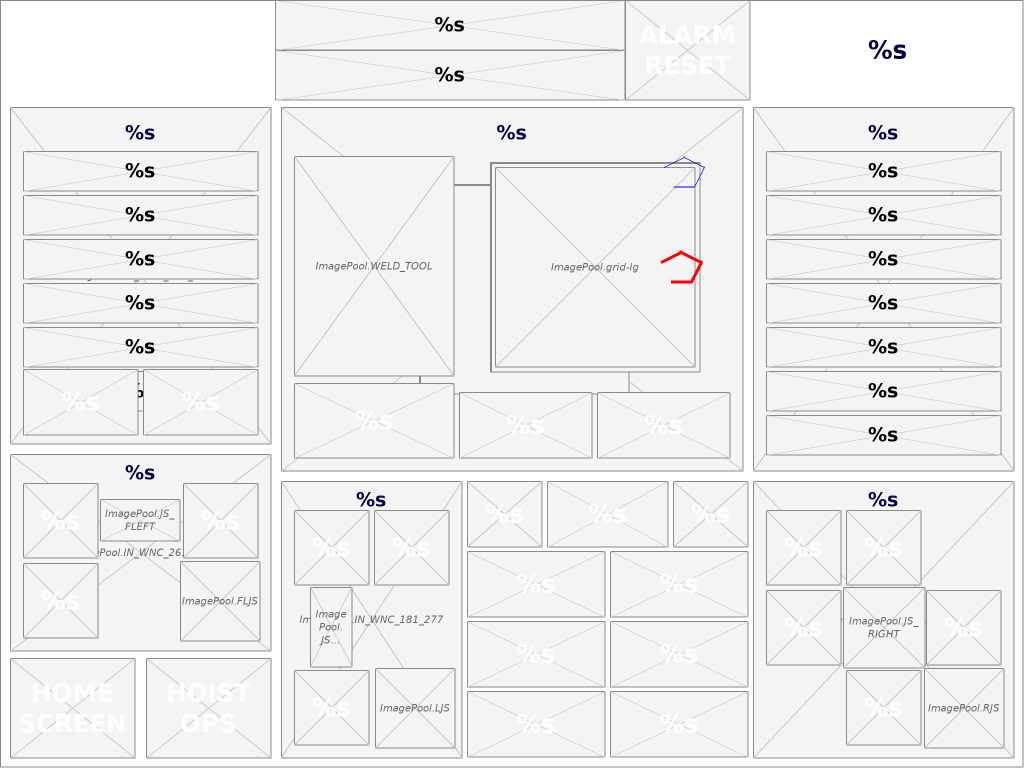
VISUALIZATION TOOL_OPS_SCREEN  // 1024x768, background image ImagePool.background1
    Image (281,107 462x364), image: ImagePool.IN_WNC_462_364
    Group (419,184 70x70), invisible if: MAIN.Visualization.P14_SMALL_PIE_DISPLAY_INVISIBLE
        Pie (1,1 209x209), invisible if: MAIN.RGP.PROG.P14_PIE_INVISIBLE[0]
        Pie (1,1 209x209), invisible if: MAIN.RGP.PROG.P14_PIE_INVISIBLE[1]
            p426801730: MAIN.RGP.PROG.P14_PIE_BEGIN[1]
            p2124672552: MAIN.RGP.PROG.P14_PIE_END[1]
        Pie (1,1 209x209), invisible if: MAIN.RGP.PROG.P14_PIE_INVISIBLE[2]
            p426801730: MAIN.RGP.PROG.P14_PIE_BEGIN[2]
            p2124672552: MAIN.RGP.PROG.P14_PIE_END[2]
        Pie (1,1 209x209), invisible if: MAIN.RGP.PROG.P14_PIE_INVISIBLE[3]
            p426801730: MAIN.RGP.PROG.P14_PIE_BEGIN[3]
            p2124672552: MAIN.RGP.PROG.P14_PIE_END[3]
        Pie (1,1 209x209), invisible if: MAIN.RGP.PROG.P14_PIE_INVISIBLE[4]
            p426801730: MAIN.RGP.PROG.P14_PIE_BEGIN[4]
            p2124672552: MAIN.RGP.PROG.P14_PIE_END[4]
        Pie (1,1 209x209), invisible if: MAIN.RGP.PROG.P14_PIE_INVISIBLE[5]
            p426801730: MAIN.RGP.PROG.P14_PIE_BEGIN[5]
            p2124672552: MAIN.RGP.PROG.P14_PIE_END[5]
        Pie (1,1 209x209), invisible if: MAIN.RGP.PROG.P14_PIE_INVISIBLE[6]
            p426801730: MAIN.RGP.PROG.P14_PIE_BEGIN[6]
            p2124672552: MAIN.RGP.PROG.P14_PIE_END[6]
        Pie (1,1 209x209), invisible if: MAIN.RGP.PROG.P14_PIE_INVISIBLE[7]
            p426801730: MAIN.RGP.PROG.P14_PIE_BEGIN[7]
            p2124672552: MAIN.RGP.PROG.P14_PIE_END[7]
        Pie (1,1 209x209), invisible if: MAIN.RGP.PROG.P14_PIE_INVISIBLE[8]
            p426801730: MAIN.RGP.PROG.P14_PIE_BEGIN[8]
            p2124672552: MAIN.RGP.PROG.P14_PIE_END[8]
        Pie (1,1 209x209), invisible if: MAIN.RGP.PROG.P14_PIE_INVISIBLE[9]
            p426801730: MAIN.RGP.PROG.P14_PIE_BEGIN[9]
            p2124672552: MAIN.RGP.PROG.P14_PIE_END[9]
        Pie (1,1 209x209), invisible if: MAIN.RGP.PROG.P14_PIE_INVISIBLE[10]
            p426801730: MAIN.RGP.PROG.P14_PIE_BEGIN[10]
            p2124672552: MAIN.RGP.PROG.P14_PIE_END[10]
        Pie (1,1 209x209), invisible if: MAIN.RGP.PROG.P14_PIE_INVISIBLE[11]
            p426801730: MAIN.RGP.PROG.P14_PIE_BEGIN[11]
            p2124672552: MAIN.RGP.PROG.P14_PIE_END[11]
        Pie (1,1 209x209), invisible if: MAIN.RGP.PROG.P14_PIE_INVISIBLE[12]
            p426801730: MAIN.RGP.PROG.P14_PIE_BEGIN[12]
            p2124672552: MAIN.RGP.PROG.P14_PIE_END[12]
        Pie (1,1 209x209), invisible if: MAIN.RGP.PROG.P14_PIE_INVISIBLE[13]
            p426801730: MAIN.RGP.PROG.P14_PIE_BEGIN[13]
            p2124672552: MAIN.RGP.PROG.P14_PIE_END[13]
        Pie (1,1 209x209), invisible if: MAIN.RGP.PROG.P14_PIE_INVISIBLE[14]
            p426801730: MAIN.RGP.PROG.P14_PIE_BEGIN[14]
            p2124672552: MAIN.RGP.PROG.P14_PIE_END[14]
        Pie (1,1 209x209), invisible if: MAIN.RGP.PROG.P14_PIE_INVISIBLE[15]
            p426801730: MAIN.RGP.PROG.P14_PIE_BEGIN[15]
            p2124672552: MAIN.RGP.PROG.P14_PIE_END[15]
        Pie (0,0 210x210), invisible if: MAIN.RGP.PROG.P14_PIE_INVISIBLE[16]
            p426801730: MAIN.RGP.PROG.P14_PIE_BEGIN[16]
            p2124672552: MAIN.RGP.PROG.P14_PIE_END[16]
        Pie (1,1 209x209), invisible if: MAIN.RGP.PROG.P14_PIE_INVISIBLE[17]
            p426801730: MAIN.RGP.PROG.P14_PIE_BEGIN[17]
            p2124672552: MAIN.RGP.PROG.P14_PIE_END[17]
        Pie (1,1 209x209), invisible if: MAIN.RGP.PROG.P14_PIE_INVISIBLE[18]
            p426801730: MAIN.RGP.PROG.P14_PIE_BEGIN[18]
            p2124672552: MAIN.RGP.PROG.P14_PIE_END[18]
        Pie (1,1 209x209), invisible if: MAIN.RGP.PROG.P14_PIE_INVISIBLE[19]
            p426801730: MAIN.RGP.PROG.P14_PIE_BEGIN[19]
            p2124672552: MAIN.RGP.PROG.P14_PIE_END[19]
        Pie (1,1 209x209), invisible if: MAIN.RGP.PROG.P14_PIE_INVISIBLE[20]
            p426801730: MAIN.RGP.PROG.P14_PIE_BEGIN[20]
            p2124672552: MAIN.RGP.PROG.P14_PIE_END[20]
        Pie (1,1 209x209), invisible if: MAIN.RGP.PROG.P14_PIE_INVISIBLE[21]
            p426801730: MAIN.RGP.PROG.P14_PIE_BEGIN[21]
            p2124672552: MAIN.RGP.PROG.P14_PIE_END[21]
        Pie (1,1 209x209), invisible if: MAIN.RGP.PROG.P14_PIE_INVISIBLE[22]
            p426801730: MAIN.RGP.PROG.P14_PIE_BEGIN[22]
            p2124672552: MAIN.RGP.PROG.P14_PIE_END[22]
        Pie (1,1 209x209), invisible if: MAIN.RGP.PROG.P14_PIE_INVISIBLE[23]
            p426801730: MAIN.RGP.PROG.P14_PIE_BEGIN[23]
            p2124672552: MAIN.RGP.PROG.P14_PIE_END[23]
        Pie (1,1 209x209), invisible if: MAIN.RGP.PROG.P14_PIE_INVISIBLE[24]
            p426801730: MAIN.RGP.PROG.P14_PIE_BEGIN[24]
            p2124672552: MAIN.RGP.PROG.P14_PIE_END[24]
        Pie (1,1 209x209), invisible if: MAIN.RGP.PROG.P14_PIE_INVISIBLE[25]
            p426801730: MAIN.RGP.PROG.P14_PIE_BEGIN[25]
            p2124672552: MAIN.RGP.PROG.P14_PIE_END[25]
        Pie (1,1 209x209), invisible if: MAIN.RGP.PROG.P14_PIE_INVISIBLE[26]
            p426801730: MAIN.RGP.PROG.P14_PIE_BEGIN[26]
            p2124672552: MAIN.RGP.PROG.P14_PIE_END[26]
        Pie (1,1 209x209), invisible if: MAIN.RGP.PROG.P14_PIE_INVISIBLE[27]
            p426801730: MAIN.RGP.PROG.P14_PIE_BEGIN[27]
            p2124672552: MAIN.RGP.PROG.P14_PIE_END[27]
        Pie (1,1 209x209), invisible if: MAIN.RGP.PROG.P14_PIE_INVISIBLE[28]
            p426801730: MAIN.RGP.PROG.P14_PIE_BEGIN[28]
            p2124672552: MAIN.RGP.PROG.P14_PIE_END[28]
        Pie (1,1 209x209), invisible if: MAIN.RGP.PROG.P14_PIE_INVISIBLE[29]
            p426801730: MAIN.RGP.PROG.P14_PIE_BEGIN[29]
            p2124672552: MAIN.RGP.PROG.P14_PIE_END[29]
        Pie (1,1 209x209), invisible if: MAIN.RGP.PROG.P14_PIE_INVISIBLE[30]
            p426801730: MAIN.RGP.PROG.P14_PIE_BEGIN[30]
            p2124672552: MAIN.RGP.PROG.P14_PIE_END[30]
        Pie (1,1 209x209), invisible if: MAIN.RGP.PROG.P14_PIE_INVISIBLE[31]
            p426801730: MAIN.RGP.PROG.P14_PIE_BEGIN[31]
            p2124672552: MAIN.RGP.PROG.P14_PIE_END[31]
        Pie (1,1 209x209), invisible if: MAIN.RGP.PROG.P14_PIE_INVISIBLE[32]
            p426801730: MAIN.RGP.PROG.P14_PIE_BEGIN[32]
            p2124672552: MAIN.RGP.PROG.P14_PIE_END[32]
        Pie (1,1 209x209), invisible if: MAIN.RGP.PROG.P14_PIE_INVISIBLE[33]
            p426801730: MAIN.RGP.PROG.P14_PIE_BEGIN[33]
            p2124672552: MAIN.RGP.PROG.P14_PIE_END[33]
        Pie (1,1 209x209), invisible if: MAIN.RGP.PROG.P14_PIE_INVISIBLE[34]
            p426801730: MAIN.RGP.PROG.P14_PIE_BEGIN[34]
            p2124672552: MAIN.RGP.PROG.P14_PIE_END[34]
        Pie (1,1 209x209), invisible if: MAIN.RGP.PROG.P14_PIE_INVISIBLE[35]
            p426801730: MAIN.RGP.PROG.P14_PIE_BEGIN[35]
            p2124672552: MAIN.RGP.PROG.P14_PIE_END[35]
        Pie (1,1 209x209), invisible if: MAIN.RGP.PROG.P14_PIE_INVISIBLE[36]
            p426801730: MAIN.RGP.PROG.P14_PIE_BEGIN[36]
            p2124672552: MAIN.RGP.PROG.P14_PIE_END[36]
        Pie (1,1 209x209), invisible if: MAIN.RGP.PROG.P14_PIE_INVISIBLE[37]
            p426801730: MAIN.RGP.PROG.P14_PIE_BEGIN[37]
            p2124672552: MAIN.RGP.PROG.P14_PIE_END[37]
        Pie (1,1 209x209), invisible if: MAIN.RGP.PROG.P14_PIE_INVISIBLE[38]
            p426801730: MAIN.RGP.PROG.P14_PIE_BEGIN[38]
            p2124672552: MAIN.RGP.PROG.P14_PIE_END[38]
        Pie (1,1 209x209), invisible if: MAIN.RGP.PROG.P14_PIE_INVISIBLE[39]
            p426801730: MAIN.RGP.PROG.P14_PIE_BEGIN[39]
            p2124672552: MAIN.RGP.PROG.P14_PIE_END[39]
        Pie (1,1 209x209), invisible if: MAIN.RGP.PROG.P14_PIE_INVISIBLE[40]
            p426801730: MAIN.RGP.PROG.P14_PIE_BEGIN[40]
            p2124672552: MAIN.RGP.PROG.P14_PIE_END[40]
        Pie (1,1 209x209), invisible if: MAIN.RGP.PROG.P14_PIE_INVISIBLE[41]
            p426801730: MAIN.RGP.PROG.P14_PIE_BEGIN[41]
            p2124672552: MAIN.RGP.PROG.P14_PIE_END[41]
        Pie (1,1 209x209), invisible if: MAIN.RGP.PROG.P14_PIE_INVISIBLE[42]
            p426801730: MAIN.RGP.PROG.P14_PIE_BEGIN[42]
            p2124672552: MAIN.RGP.PROG.P14_PIE_END[42]
        Pie (1,1 209x209), invisible if: MAIN.RGP.PROG.P14_PIE_INVISIBLE[43]
            p426801730: MAIN.RGP.PROG.P14_PIE_BEGIN[43]
            p2124672552: MAIN.RGP.PROG.P14_PIE_END[43]
        Pie (1,1 209x209), invisible if: MAIN.RGP.PROG.P14_PIE_INVISIBLE[44]
            p426801730: MAIN.RGP.PROG.P14_PIE_BEGIN[44]
            p2124672552: MAIN.RGP.PROG.P14_PIE_END[44]
        Pie (1,1 209x209), invisible if: MAIN.RGP.PROG.P14_PIE_INVISIBLE[45]
            p426801730: MAIN.RGP.PROG.P14_PIE_BEGIN[45]
            p2124672552: MAIN.RGP.PROG.P14_PIE_END[45]
        Pie (1,1 209x209), invisible if: MAIN.RGP.PROG.P14_PIE_INVISIBLE[46]
            p426801730: MAIN.RGP.PROG.P14_PIE_BEGIN[46]
            p2124672552: MAIN.RGP.PROG.P14_PIE_END[46]
        Pie (1,1 209x209), invisible if: MAIN.RGP.PROG.P14_PIE_INVISIBLE[47]
            p426801730: MAIN.RGP.PROG.P14_PIE_BEGIN[47]
            p2124672552: MAIN.RGP.PROG.P14_PIE_END[47]
        Pie (1,1 209x209), invisible if: MAIN.RGP.PROG.P14_PIE_INVISIBLE[48]
            p426801730: MAIN.RGP.PROG.P14_PIE_BEGIN[48]
            p2124672552: MAIN.RGP.PROG.P14_PIE_END[48]
        Pie (1,1 209x209), invisible if: MAIN.RGP.PROG.P14_PIE_INVISIBLE[49]
            p426801730: MAIN.RGP.PROG.P14_PIE_BEGIN[49]
            p2124672552: MAIN.RGP.PROG.P14_PIE_END[49]
        Pie (1,1 209x209), invisible if: MAIN.RGP.PROG.P14_PIE_INVISIBLE[50]
            p426801730: MAIN.RGP.PROG.P14_PIE_BEGIN[50]
            p2124672552: MAIN.RGP.PROG.P14_PIE_END[50]
        Pie (1,1 209x209), invisible if: MAIN.RGP.PROG.P14_PIE_INVISIBLE[0]
        Pie (1,1 209x209), invisible if: MAIN.RGP.PROG.P14_PIE_INVISIBLE[0]
            p426801730: MAIN.RGP.PROG.P14_PIE_BEGIN[0]
            p2124672552: MAIN.RGP.PROG.P14_PIE_END[0]
    Group (490,162 210x210), invisible if: MAIN.Visualization.P14_LARGE_PIE_DISPLAY_INVISIBLE
        Pie (1,1 209x209), invisible if: MAIN.RGP.PROG.P14_PIE_INVISIBLE[0]
        Pie (1,1 209x209), invisible if: MAIN.RGP.PROG.P14_PIE_INVISIBLE[1]
            p426801730: MAIN.RGP.PROG.P14_PIE_BEGIN[1]
            p2124672552: MAIN.RGP.PROG.P14_PIE_END[1]
        Pie (1,1 209x209), invisible if: MAIN.RGP.PROG.P14_PIE_INVISIBLE[2]
            p426801730: MAIN.RGP.PROG.P14_PIE_BEGIN[2]
            p2124672552: MAIN.RGP.PROG.P14_PIE_END[2]
        Pie (1,1 209x209), invisible if: MAIN.RGP.PROG.P14_PIE_INVISIBLE[3]
            p426801730: MAIN.RGP.PROG.P14_PIE_BEGIN[3]
            p2124672552: MAIN.RGP.PROG.P14_PIE_END[3]
        Pie (1,1 209x209), invisible if: MAIN.RGP.PROG.P14_PIE_INVISIBLE[4]
            p426801730: MAIN.RGP.PROG.P14_PIE_BEGIN[4]
            p2124672552: MAIN.RGP.PROG.P14_PIE_END[4]
        Pie (1,1 209x209), invisible if: MAIN.RGP.PROG.P14_PIE_INVISIBLE[5]
            p426801730: MAIN.RGP.PROG.P14_PIE_BEGIN[5]
            p2124672552: MAIN.RGP.PROG.P14_PIE_END[5]
        Pie (1,1 209x209), invisible if: MAIN.RGP.PROG.P14_PIE_INVISIBLE[6]
            p426801730: MAIN.RGP.PROG.P14_PIE_BEGIN[6]
            p2124672552: MAIN.RGP.PROG.P14_PIE_END[6]
        Pie (1,1 209x209), invisible if: MAIN.RGP.PROG.P14_PIE_INVISIBLE[7]
            p426801730: MAIN.RGP.PROG.P14_PIE_BEGIN[7]
            p2124672552: MAIN.RGP.PROG.P14_PIE_END[7]
        Pie (1,1 209x209), invisible if: MAIN.RGP.PROG.P14_PIE_INVISIBLE[8]
            p426801730: MAIN.RGP.PROG.P14_PIE_BEGIN[8]
            p2124672552: MAIN.RGP.PROG.P14_PIE_END[8]
        Pie (1,1 209x209), invisible if: MAIN.RGP.PROG.P14_PIE_INVISIBLE[9]
            p426801730: MAIN.RGP.PROG.P14_PIE_BEGIN[9]
            p2124672552: MAIN.RGP.PROG.P14_PIE_END[9]
        Pie (1,1 209x209), invisible if: MAIN.RGP.PROG.P14_PIE_INVISIBLE[10]
            p426801730: MAIN.RGP.PROG.P14_PIE_BEGIN[10]
            p2124672552: MAIN.RGP.PROG.P14_PIE_END[10]
        Pie (1,1 209x209), invisible if: MAIN.RGP.PROG.P14_PIE_INVISIBLE[11]
            p426801730: MAIN.RGP.PROG.P14_PIE_BEGIN[11]
            p2124672552: MAIN.RGP.PROG.P14_PIE_END[11]
        Pie (1,1 209x209), invisible if: MAIN.RGP.PROG.P14_PIE_INVISIBLE[12]
            p426801730: MAIN.RGP.PROG.P14_PIE_BEGIN[12]
            p2124672552: MAIN.RGP.PROG.P14_PIE_END[12]
        Pie (1,1 209x209), invisible if: MAIN.RGP.PROG.P14_PIE_INVISIBLE[13]
            p426801730: MAIN.RGP.PROG.P14_PIE_BEGIN[13]
            p2124672552: MAIN.RGP.PROG.P14_PIE_END[13]
        Pie (1,1 209x209), invisible if: MAIN.RGP.PROG.P14_PIE_INVISIBLE[14]
            p426801730: MAIN.RGP.PROG.P14_PIE_BEGIN[14]
            p2124672552: MAIN.RGP.PROG.P14_PIE_END[14]
        Pie (1,1 209x209), invisible if: MAIN.RGP.PROG.P14_PIE_INVISIBLE[15]
            p426801730: MAIN.RGP.PROG.P14_PIE_BEGIN[15]
            p2124672552: MAIN.RGP.PROG.P14_PIE_END[15]
        Pie (0,0 210x210), invisible if: MAIN.RGP.PROG.P14_PIE_INVISIBLE[16]
            p426801730: MAIN.RGP.PROG.P14_PIE_BEGIN[16]
            p2124672552: MAIN.RGP.PROG.P14_PIE_END[16]
        Pie (1,1 209x209), invisible if: MAIN.RGP.PROG.P14_PIE_INVISIBLE[17]
            p426801730: MAIN.RGP.PROG.P14_PIE_BEGIN[17]
            p2124672552: MAIN.RGP.PROG.P14_PIE_END[17]
        Pie (1,1 209x209), invisible if: MAIN.RGP.PROG.P14_PIE_INVISIBLE[18]
            p426801730: MAIN.RGP.PROG.P14_PIE_BEGIN[18]
            p2124672552: MAIN.RGP.PROG.P14_PIE_END[18]
        Pie (1,1 209x209), invisible if: MAIN.RGP.PROG.P14_PIE_INVISIBLE[19]
            p426801730: MAIN.RGP.PROG.P14_PIE_BEGIN[19]
            p2124672552: MAIN.RGP.PROG.P14_PIE_END[19]
        Pie (1,1 209x209), invisible if: MAIN.RGP.PROG.P14_PIE_INVISIBLE[20]
            p426801730: MAIN.RGP.PROG.P14_PIE_BEGIN[20]
            p2124672552: MAIN.RGP.PROG.P14_PIE_END[20]
        Pie (1,1 209x209), invisible if: MAIN.RGP.PROG.P14_PIE_INVISIBLE[21]
            p426801730: MAIN.RGP.PROG.P14_PIE_BEGIN[21]
            p2124672552: MAIN.RGP.PROG.P14_PIE_END[21]
        Pie (1,1 209x209), invisible if: MAIN.RGP.PROG.P14_PIE_INVISIBLE[22]
            p426801730: MAIN.RGP.PROG.P14_PIE_BEGIN[22]
            p2124672552: MAIN.RGP.PROG.P14_PIE_END[22]
        Pie (1,1 209x209), invisible if: MAIN.RGP.PROG.P14_PIE_INVISIBLE[23]
            p426801730: MAIN.RGP.PROG.P14_PIE_BEGIN[23]
            p2124672552: MAIN.RGP.PROG.P14_PIE_END[23]
        Pie (1,1 209x209), invisible if: MAIN.RGP.PROG.P14_PIE_INVISIBLE[24]
            p426801730: MAIN.RGP.PROG.P14_PIE_BEGIN[24]
            p2124672552: MAIN.RGP.PROG.P14_PIE_END[24]
        Pie (1,1 209x209), invisible if: MAIN.RGP.PROG.P14_PIE_INVISIBLE[25]
            p426801730: MAIN.RGP.PROG.P14_PIE_BEGIN[25]
            p2124672552: MAIN.RGP.PROG.P14_PIE_END[25]
        Pie (1,1 209x209), invisible if: MAIN.RGP.PROG.P14_PIE_INVISIBLE[26]
            p426801730: MAIN.RGP.PROG.P14_PIE_BEGIN[26]
            p2124672552: MAIN.RGP.PROG.P14_PIE_END[26]
        Pie (1,1 209x209), invisible if: MAIN.RGP.PROG.P14_PIE_INVISIBLE[27]
            p426801730: MAIN.RGP.PROG.P14_PIE_BEGIN[27]
            p2124672552: MAIN.RGP.PROG.P14_PIE_END[27]
        Pie (1,1 209x209), invisible if: MAIN.RGP.PROG.P14_PIE_INVISIBLE[28]
            p426801730: MAIN.RGP.PROG.P14_PIE_BEGIN[28]
            p2124672552: MAIN.RGP.PROG.P14_PIE_END[28]
        Pie (1,1 209x209), invisible if: MAIN.RGP.PROG.P14_PIE_INVISIBLE[29]
            p426801730: MAIN.RGP.PROG.P14_PIE_BEGIN[29]
            p2124672552: MAIN.RGP.PROG.P14_PIE_END[29]
        Pie (1,1 209x209), invisible if: MAIN.RGP.PROG.P14_PIE_INVISIBLE[30]
            p426801730: MAIN.RGP.PROG.P14_PIE_BEGIN[30]
            p2124672552: MAIN.RGP.PROG.P14_PIE_END[30]
        Pie (1,1 209x209), invisible if: MAIN.RGP.PROG.P14_PIE_INVISIBLE[31]
            p426801730: MAIN.RGP.PROG.P14_PIE_BEGIN[31]
            p2124672552: MAIN.RGP.PROG.P14_PIE_END[31]
        Pie (1,1 209x209), invisible if: MAIN.RGP.PROG.P14_PIE_INVISIBLE[32]
            p426801730: MAIN.RGP.PROG.P14_PIE_BEGIN[32]
            p2124672552: MAIN.RGP.PROG.P14_PIE_END[32]
        Pie (1,1 209x209), invisible if: MAIN.RGP.PROG.P14_PIE_INVISIBLE[33]
            p426801730: MAIN.RGP.PROG.P14_PIE_BEGIN[33]
            p2124672552: MAIN.RGP.PROG.P14_PIE_END[33]
        Pie (1,1 209x209), invisible if: MAIN.RGP.PROG.P14_PIE_INVISIBLE[34]
            p426801730: MAIN.RGP.PROG.P14_PIE_BEGIN[34]
            p2124672552: MAIN.RGP.PROG.P14_PIE_END[34]
        Pie (1,1 209x209), invisible if: MAIN.RGP.PROG.P14_PIE_INVISIBLE[35]
            p426801730: MAIN.RGP.PROG.P14_PIE_BEGIN[35]
            p2124672552: MAIN.RGP.PROG.P14_PIE_END[35]
        Pie (1,1 209x209), invisible if: MAIN.RGP.PROG.P14_PIE_INVISIBLE[36]
            p426801730: MAIN.RGP.PROG.P14_PIE_BEGIN[36]
            p2124672552: MAIN.RGP.PROG.P14_PIE_END[36]
        Pie (1,1 209x209), invisible if: MAIN.RGP.PROG.P14_PIE_INVISIBLE[37]
            p426801730: MAIN.RGP.PROG.P14_PIE_BEGIN[37]
            p2124672552: MAIN.RGP.PROG.P14_PIE_END[37]
        Pie (1,1 209x209), invisible if: MAIN.RGP.PROG.P14_PIE_INVISIBLE[38]
            p426801730: MAIN.RGP.PROG.P14_PIE_BEGIN[38]
            p2124672552: MAIN.RGP.PROG.P14_PIE_END[38]
        Pie (1,1 209x209), invisible if: MAIN.RGP.PROG.P14_PIE_INVISIBLE[39]
            p426801730: MAIN.RGP.PROG.P14_PIE_BEGIN[39]
            p2124672552: MAIN.RGP.PROG.P14_PIE_END[39]
        Pie (1,1 209x209), invisible if: MAIN.RGP.PROG.P14_PIE_INVISIBLE[40]
            p426801730: MAIN.RGP.PROG.P14_PIE_BEGIN[40]
            p2124672552: MAIN.RGP.PROG.P14_PIE_END[40]
        Pie (1,1 209x209), invisible if: MAIN.RGP.PROG.P14_PIE_INVISIBLE[41]
            p426801730: MAIN.RGP.PROG.P14_PIE_BEGIN[41]
            p2124672552: MAIN.RGP.PROG.P14_PIE_END[41]
        Pie (1,1 209x209), invisible if: MAIN.RGP.PROG.P14_PIE_INVISIBLE[42]
            p426801730: MAIN.RGP.PROG.P14_PIE_BEGIN[42]
            p2124672552: MAIN.RGP.PROG.P14_PIE_END[42]
        Pie (1,1 209x209), invisible if: MAIN.RGP.PROG.P14_PIE_INVISIBLE[43]
            p426801730: MAIN.RGP.PROG.P14_PIE_BEGIN[43]
            p2124672552: MAIN.RGP.PROG.P14_PIE_END[43]
        Pie (1,1 209x209), invisible if: MAIN.RGP.PROG.P14_PIE_INVISIBLE[44]
            p426801730: MAIN.RGP.PROG.P14_PIE_BEGIN[44]
            p2124672552: MAIN.RGP.PROG.P14_PIE_END[44]
        Pie (1,1 209x209), invisible if: MAIN.RGP.PROG.P14_PIE_INVISIBLE[45]
            p426801730: MAIN.RGP.PROG.P14_PIE_BEGIN[45]
            p2124672552: MAIN.RGP.PROG.P14_PIE_END[45]
        Pie (1,1 209x209), invisible if: MAIN.RGP.PROG.P14_PIE_INVISIBLE[46]
            p426801730: MAIN.RGP.PROG.P14_PIE_BEGIN[46]
            p2124672552: MAIN.RGP.PROG.P14_PIE_END[46]
        Pie (1,1 209x209), invisible if: MAIN.RGP.PROG.P14_PIE_INVISIBLE[47]
            p426801730: MAIN.RGP.PROG.P14_PIE_BEGIN[47]
            p2124672552: MAIN.RGP.PROG.P14_PIE_END[47]
        Pie (1,1 209x209), invisible if: MAIN.RGP.PROG.P14_PIE_INVISIBLE[48]
            p426801730: MAIN.RGP.PROG.P14_PIE_BEGIN[48]
            p2124672552: MAIN.RGP.PROG.P14_PIE_END[48]
        Pie (1,1 209x209), invisible if: MAIN.RGP.PROG.P14_PIE_INVISIBLE[49]
            p426801730: MAIN.RGP.PROG.P14_PIE_BEGIN[49]
            p2124672552: MAIN.RGP.PROG.P14_PIE_END[49]
        Pie (1,1 209x209), invisible if: MAIN.RGP.PROG.P14_PIE_INVISIBLE[50]
            p426801730: MAIN.RGP.PROG.P14_PIE_BEGIN[50]
            p2124672552: MAIN.RGP.PROG.P14_PIE_END[50]
        Pie (1,1 209x209), invisible if: MAIN.RGP.PROG.P14_PIE_INVISIBLE[0]
        Pie (1,1 209x209), invisible if: MAIN.RGP.PROG.P14_PIE_INVISIBLE[0]
            p426801730: MAIN.RGP.PROG.P14_PIE_BEGIN[0]
            p2124672552: MAIN.RGP.PROG.P14_PIE_END[0]
    Image (495,167 200x200), invisible if: MAIN.Visualization.P14_Profile.invisible, image: ImagePool.grid-lg
    Image (10,454 261x197), image: ImagePool.IN_WNC_261_197
    Image (23,563 75x75), "%s", text variable: MAIN.Visualization.P14_JSFARLEFT_SP.display_text, invisible if: MAIN.Visualization.P14_JSFARLEFT_SP.invisible, image: ImagePool.PB_BU_75_75
        p84334746: MAIN.Visualization.P14_JSFARLEFT_SP.bitmap_ID
        OnMouseDown: execute { MAIN.Visualization.P14_JSFARLEFT_SP.Active:=TRUE; }
        OnMouseUp: execute { MAIN.Visualization.P14_JSFARLEFT_SP.Active:=FALSE; }
    Image (23,483 75x75), "%s", text variable: MAIN.Visualization.P14_JSFARLEFT_LT.display_text, invisible if: MAIN.Visualization.P14_JSFARLEFT_LT.invisible, image: ImagePool.PB_BU_75_75
        p84334746: MAIN.Visualization.P14_JSFARLEFT_LT.bitmap_ID
        OnMouseDown: execute { MAIN.Visualization.P14_JSFARLEFT_LT.Active:=TRUE; }
        OnMouseUp: execute { MAIN.Visualization.P14_JSFARLEFT_LT.Active:=FALSE; }
    Image (100,499 80x42), image: ImagePool.JS_FLEFT
    Image (183,483 75x75), "%s", text variable: MAIN.Visualization.P14_JSFARLEFT_RT.display_text, invisible if: MAIN.Visualization.P14_JSFARLEFT_RT.invisible, image: ImagePool.PB_BU_75_75
        p84334746: MAIN.Visualization.P14_JSFARLEFT_RT.bitmap_ID
        OnMouseDown: execute { MAIN.Visualization.P14_JSFARLEFT_RT.Active:=TRUE; }
        OnMouseUp: execute { MAIN.Visualization.P14_JSFARLEFT_RT.Active:=FALSE; }
    Image (180,561 80x80), image: ImagePool.FLJS
    Textfield (10,458 261x30), "%s", text variable: MAIN.Visualization.P14_JSFARLEFT_DISP.display_text
        OnMouseDown: execute { MAIN.Visualization.P14_JSFARLEFT_DISP.Active:=TRUE; }
        OnMouseUp: execute { MAIN.Visualization.P14_JSFARLEFT_DISP.Active:=FALSE; }
    Textfield (750,0 275x100), "%s", text variable: MAIN.Visualization.P00D_Active_Panel.display_text
    Image (275,0 350x50), "%s", text variable: MAIN.Visualization.P00D_Station_Status.display_text, image: ImagePool.IN_BU_300_50
        p84334746: MAIN.Visualization.P00D_Station_Status.bitmap_ID
    Image (625,0 125x100), "ALARM RESET", image: ImagePool.PB_BU_125_100
        p84334746: MAIN.Visualization.P00B_Alarm_Reset.bitmap_ID
        OnMouseDown: execute { MAIN.Visualization.P00B_Alarm_Reset.Active:=TRUE; }
        OnMouseUp: execute { MAIN.Visualization.P00B_Alarm_Reset.Active:=FALSE; }
    Image (275,50 350x50), "%s", text variable: MAIN.Visualization.P00D_Alarm_Status.display_text, image: ImagePool.IN_BU_300_50
        p84334746: MAIN.Visualization.P00D_Alarm_Status.bitmap_ID
    Image (10,658 125x100), "HOME SCREEN", image: ImagePool.PB_BU_125_100
        OnMouseDown: execute { MAIN.Visualization.P14_Home_Screen.Active:=TRUE; }
        OnMouseUp: execute { MAIN.Visualization.P14_Home_Screen.Active:=FALSE; }
    Image (753,107 261x364), image: ImagePool.IN_WNC_261_364
    Textfield (753,115 261x36), "%s", text variable: MAIN.Visualization.P14_DISP_1.display_text
        OnMouseDown: execute { MAIN.Visualization.P14_DISP_1.Active:=TRUE; }
        OnMouseUp: execute { MAIN.Visualization.P14_DISP_1.Active:=FALSE; }
    Image (766,151 235x40), "%s", text variable: MAIN.Visualization.P14_DISP_2.display_text, invisible if: MAIN.Visualization.P14_DISP_2.invisible, image: ImagePool.IN_BU_300_50
        p84334746: MAIN.Visualization.P14_DISP_2.bitmap_ID
    Image (766,195 235x40), "%s", text variable: MAIN.Visualization.P14_DISP_3.display_text, invisible if: MAIN.Visualization.P14_DISP_3.invisible, image: ImagePool.IN_BU_300_50
        p84334746: MAIN.Visualization.P14_DISP_3.bitmap_ID
    Image (766,239 235x40), "%s", text variable: MAIN.Visualization.P14_DISP_4.display_text, invisible if: MAIN.Visualization.P14_DISP_4.invisible, image: ImagePool.IN_BU_300_50
        p84334746: MAIN.Visualization.P14_DISP_4.bitmap_ID
    Image (766,283 235x40), "%s", text variable: MAIN.Visualization.P14_DISP_5.display_text, invisible if: MAIN.Visualization.P14_DISP_5.invisible, image: ImagePool.IN_BU_300_50
        p84334746: MAIN.Visualization.P14_DISP_5.bitmap_ID
    Image (766,327 235x40), "%s", text variable: MAIN.Visualization.P14_DISP_6.display_text, invisible if: MAIN.Visualization.P14_DISP_6.invisible, image: ImagePool.IN_BU_300_50
        p84334746: MAIN.Visualization.P14_DISP_6.bitmap_ID
    Image (766,371 235x40), "%s", text variable: MAIN.Visualization.P14_DISP_7.display_text, invisible if: MAIN.Visualization.P14_DISP_7.invisible, image: ImagePool.IN_BU_300_50
        p84334746: MAIN.Visualization.P14_DISP_7.bitmap_ID
    Image (753,481 261x277), image: ImagePool.IN_WNC_261_277
    Image (846,510 75x75), "%s", text variable: MAIN.Visualization.P14_JSRIGHT_UP.display_text, invisible if: MAIN.Visualization.P14_JSRIGHT_UP.invisible, image: ImagePool.PB_BU_75_75
        p84334746: MAIN.Visualization.P14_JSRIGHT_UP.bitmap_ID
        OnMouseDown: execute { MAIN.Visualization.P14_JSRIGHT_UP.Active:=TRUE; }
        OnMouseUp: execute { MAIN.Visualization.P14_JSRIGHT_UP.Active:=FALSE; }
    Image (766,510 75x75), "%s", text variable: MAIN.Visualization.P14_JSRIGHT_SP.display_text, invisible if: MAIN.Visualization.P14_JSRIGHT_SP.invisible, image: ImagePool.PB_BU_75_75
        p84334746: MAIN.Visualization.P14_JSRIGHT_SP.bitmap_ID
        OnMouseDown: execute { MAIN.Visualization.P14_JSRIGHT_SP.Active:=TRUE; }
        OnMouseUp: execute { MAIN.Visualization.P14_JSRIGHT_SP.Active:=FALSE; }
    Image (766,590 75x75), "%s", text variable: MAIN.Visualization.P14_JSRIGHT_LT.display_text, invisible if: MAIN.Visualization.P14_JSRIGHT_LT.invisible, image: ImagePool.PB_BU_75_75
        p84334746: MAIN.Visualization.P14_JSRIGHT_LT.bitmap_ID
        OnMouseDown: execute { MAIN.Visualization.P14_JSRIGHT_LT.Active:=TRUE; }
        OnMouseUp: execute { MAIN.Visualization.P14_JSRIGHT_LT.Active:=FALSE; }
    Image (843,587 82x81), image: ImagePool.JS_RIGHT
    Image (926,590 75x75), "%s", text variable: MAIN.Visualization.P14_JSRIGHT_RT.display_text, invisible if: MAIN.Visualization.P14_JSRIGHT_RT.invisible, image: ImagePool.PB_BU_75_75
        p84334746: MAIN.Visualization.P14_JSRIGHT_RT.bitmap_ID
        OnMouseDown: execute { MAIN.Visualization.P14_JSRIGHT_RT.Active:=TRUE; }
        OnMouseUp: execute { MAIN.Visualization.P14_JSRIGHT_RT.Active:=FALSE; }
    Image (846,670 75x75), "%s", text variable: MAIN.Visualization.P14_JSRIGHT_DN.display_text, invisible if: MAIN.Visualization.P14_JSRIGHT_DN.invisible, image: ImagePool.PB_BU_75_75
        p84334746: MAIN.Visualization.P14_JSRIGHT_DN.bitmap_ID
        OnMouseDown: execute { MAIN.Visualization.P14_JSRIGHT_DN.Active:=TRUE; }
        OnMouseUp: execute { MAIN.Visualization.P14_JSRIGHT_DN.Active:=FALSE; }
    Textfield (753,485 261x30), "%s", text variable: MAIN.Visualization.P14_JSRIGHT_DISP.display_text
        OnMouseDown: execute { MAIN.Visualization.P14_JSRIGHT_DISP.Active:=TRUE; }
        OnMouseUp: execute { MAIN.Visualization.P14_JSRIGHT_DISP.Active:=FALSE; }
    Image (281,481 181x277), image: ImagePool.IN_WNC_181_277
    Image (294,510 75x75), "%s", text variable: MAIN.Visualization.P14_JSLEFT_UP.display_text, invisible if: MAIN.Visualization.P14_JSLEFT_UP.invisible, image: ImagePool.PB_BU_75_75
        p84334746: MAIN.Visualization.P14_JSLEFT_UP.bitmap_ID
        OnMouseDown: execute { MAIN.Visualization.P14_JSLEFT_UP.Active:=TRUE; }
        OnMouseUp: execute { MAIN.Visualization.P14_JSLEFT_UP.Active:=FALSE; }
    Image (374,510 75x75), "%s", text variable: MAIN.Visualization.P14_JSLEFT_SP.display_text, invisible if: MAIN.Visualization.P14_JSLEFT_SP.invisible, image: ImagePool.PB_BU_75_75
        p84334746: MAIN.Visualization.P14_JSLEFT_SP.bitmap_ID
        OnMouseDown: execute { MAIN.Visualization.P14_JSLEFT_SP.Active:=TRUE; }
        OnMouseUp: execute { MAIN.Visualization.P14_JSLEFT_SP.Active:=FALSE; }
    Image (310,587 42x80), image: ImagePool.JS_LEFT
    Image (294,670 75x75), "%s", text variable: MAIN.Visualization.P14_JSLEFT_DN.display_text, invisible if: MAIN.Visualization.P14_JSLEFT_DN.invisible, image: ImagePool.PB_BU_75_75
        p84334746: MAIN.Visualization.P14_JSLEFT_DN.bitmap_ID
        OnMouseDown: execute { MAIN.Visualization.P14_JSLEFT_DN.Active:=TRUE; }
        OnMouseUp: execute { MAIN.Visualization.P14_JSLEFT_DN.Active:=FALSE; }
    Textfield (281,485 181x30), "%s", text variable: MAIN.Visualization.P14_JSLEFT_DISP.display_text
        OnMouseDown: execute { MAIN.Visualization.P14_JSLEFT_DISP.Active:=TRUE; }
        OnMouseUp: execute { MAIN.Visualization.P14_JSLEFT_DISP.Active:=FALSE; }
    Image (146,658 125x100), "HOIST OPS", image: ImagePool.PB_BU_125_100
        p84334746: MAIN.Visualization.P14_Hoist_Ops.bitmap_ID
        OnMouseDown: execute { MAIN.Visualization.P14_Hoist_Ops.Active:=TRUE; }
        OnMouseUp: execute { MAIN.Visualization.P14_Hoist_Ops.Active:=FALSE; }
    Image (766,415 235x40), "%s", text variable: MAIN.Visualization.P14_DISP_8.display_text, invisible if: MAIN.Visualization.P14_DISP_8.invisible, image: ImagePool.IN_BU_300_50
        p84334746: MAIN.Visualization.P14_DISP_8.bitmap_ID
    Image (467,691 138x66), "%s", text variable: MAIN.Visualization.P14_Button_3.display_text, invisible if: MAIN.Visualization.P14_Button_3.invisible, image: ImagePool.PB_BU_160_75
        p84334746: MAIN.Visualization.P14_Button_3.bitmap_ID
        OnMouseDown: execute { MAIN.Visualization.P14_Button_3.Active:=TRUE; }
        OnMouseUp: execute { MAIN.Visualization.P14_Button_3.Active:=FALSE; }
    Image (610,691 138x66), "%s", text variable: MAIN.Visualization.P14_Button_4.display_text, invisible if: MAIN.Visualization.P14_Button_4.invisible, image: ImagePool.PB_BU_160_75
        p84334746: MAIN.Visualization.P14_Button_4.bitmap_ID
        OnMouseDown: execute { MAIN.Visualization.P14_Button_4.Active:=TRUE; }
        OnMouseUp: execute { MAIN.Visualization.P14_Button_4.Active:=FALSE; }
    Image (467,621 138x66), "%s", text variable: MAIN.Visualization.P14_Button_1.display_text, invisible if: MAIN.Visualization.P14_Button_1.invisible, image: ImagePool.PB_BU_160_75
        p84334746: MAIN.Visualization.P14_Button_1.bitmap_ID
        OnMouseDown: execute { MAIN.Visualization.P14_Button_1.Active:=TRUE; }
        OnMouseUp: execute { MAIN.Visualization.P14_Button_1.Active:=FALSE; }
    Image (610,621 138x66), "%s", text variable: MAIN.Visualization.P14_Button_2.display_text, invisible if: MAIN.Visualization.P14_Button_2.invisible, image: ImagePool.PB_BU_160_75
        p84334746: MAIN.Visualization.P14_Button_2.bitmap_ID
        OnMouseDown: execute { MAIN.Visualization.P14_Button_2.Active:=TRUE; }
        OnMouseUp: execute { MAIN.Visualization.P14_Button_2.Active:=FALSE; }
    Image (10,107 261x337), image: ImagePool.IN_WNC_261_364
    Textfield (10,115 261x36), "%s", text variable: MAIN.Visualization.P14_LDISP_1.display_text
        OnMouseDown: execute { MAIN.Visualization.P14_LDISP_1.Active:=TRUE; }
        OnMouseUp: execute { MAIN.Visualization.P14_LDISP_1.Active:=FALSE; }
    Image (23,151 235x40), "%s", text variable: MAIN.Visualization.P14_LDISP_2.display_text, invisible if: MAIN.Visualization.P14_LDISP_2.invisible, image: ImagePool.IN_BU_300_50
        p84334746: MAIN.Visualization.P14_LDISP_2.bitmap_ID
    Image (23,195 235x40), "%s", text variable: MAIN.Visualization.P14_LDISP_3.display_text, invisible if: MAIN.Visualization.P14_LDISP_3.invisible, image: ImagePool.IN_BU_300_50
        p84334746: MAIN.Visualization.P14_LDISP_3.bitmap_ID
    Image (23,239 235x40), "%s", text variable: MAIN.Visualization.P14_LDISP_4.display_text, invisible if: MAIN.Visualization.P14_LDISP_4.invisible, image: ImagePool.IN_BU_300_50
        p84334746: MAIN.Visualization.P14_LDISP_4.bitmap_ID
    Image (23,283 235x40), "%s", text variable: MAIN.Visualization.P14_LDISP_5.display_text, invisible if: MAIN.Visualization.P14_LDISP_5.invisible, image: ImagePool.IN_BU_300_50
        p84334746: MAIN.Visualization.P14_LDISP_5.bitmap_ID
    Image (23,327 235x40), "%s", text variable: MAIN.Visualization.P14_LDISP_6.display_text, invisible if: MAIN.Visualization.P14_LDISP_6.invisible, image: ImagePool.IN_BU_300_50
        p84334746: MAIN.Visualization.P14_LDISP_6.bitmap_ID
    Image (23,371 235x40), "%s", text variable: MAIN.Visualization.P14_LDISP_7.display_text, invisible if: MAIN.Visualization.P14_LDISP_7.invisible, image: ImagePool.IN_BU_300_50
        p84334746: MAIN.Visualization.P14_LDISP_7.bitmap_ID
    Image (467,481 75x66), "%s", text variable: MAIN.Visualization.P14_CButton_1.display_text, invisible if: MAIN.Visualization.P14_CButton_1.invisible, image: ImagePool.PB_BU_75_75
        p84334746: MAIN.Visualization.P14_CButton_1.bitmap_ID
        OnMouseDown: execute { MAIN.Visualization.P14_CButton_1.Active:=TRUE; }
        OnMouseUp: execute { MAIN.Visualization.P14_CButton_1.Active:=FALSE; }
    Image (547,481 121x66), "%s", text variable: MAIN.Visualization.P14_CButton_3.display_text, invisible if: MAIN.Visualization.P14_CButton_3.invisible, image: ImagePool.PB_BU_160_75
        p84334746: MAIN.Visualization.P14_CButton_3.bitmap_ID
        OnMouseDown: execute { MAIN.Visualization.P14_CButton_3.Active:=TRUE; }
        OnMouseDown: write MAIN.Visualization.P14_Entered_Speed via VisuDialogs.Numpad, min MAIN.RGP.PROG.P14_ROT_SPEED_MIN, max MAIN.RGP.PROG.P14_ROT_SPEED_MAX
        OnMouseUp: execute { MAIN.Visualization.P14_CButton_3.Active:=FALSE; }
    Image (673,481 75x66), "%s", text variable: MAIN.Visualization.P14_CButton_5.display_text, invisible if: MAIN.Visualization.P14_CButton_5.invisible, image: ImagePool.PB_BU_75_75
        p84334746: MAIN.Visualization.P14_CButton_5.bitmap_ID
        OnMouseDown: execute { MAIN.Visualization.P14_CButton_5.Active:=TRUE; }
        OnMouseUp: execute { MAIN.Visualization.P14_CButton_5.Active:=FALSE; }
    Image (467,551 138x66), "%s", text variable: MAIN.Visualization.P14_CButton_6.display_text, invisible if: MAIN.Visualization.P14_CButton_6.invisible, image: ImagePool.PB_BU_160_75
        p84334746: MAIN.Visualization.P14_CButton_6.bitmap_ID
        OnMouseDown: execute { MAIN.Visualization.P14_CButton_6.Active:=TRUE; }
        OnMouseUp: execute { MAIN.Visualization.P14_CButton_6.Active:=FALSE; }
    Image (610,551 138x66), "%s", text variable: MAIN.Visualization.P14_CButton_8.display_text, invisible if: MAIN.Visualization.P14_CButton_8.invisible, image: ImagePool.PB_BU_160_75
        p84334746: MAIN.Visualization.P14_CButton_8.bitmap_ID
        OnMouseDown: execute { MAIN.Visualization.P14_CButton_8.Active:=TRUE; }
        OnMouseUp: execute { MAIN.Visualization.P14_CButton_8.Active:=FALSE; }
    Image (294,383 160x75), "%s", text variable: MAIN.Visualization.P14_CButton_7.display_text, invisible if: MAIN.Visualization.P14_CButton_7.invisible, image: ImagePool.PB_BU_160_75
        p84334746: MAIN.Visualization.P14_CButton_7.bitmap_ID
        OnMouseDown: execute { MAIN.Visualization.P14_CButton_7.Active:=TRUE; }
        OnMouseUp: execute { MAIN.Visualization.P14_CButton_7.Active:=FALSE; }
    Textfield (281,115 462x36), "%s", text variable: MAIN.Visualization.P14_CDISP.display_text
        OnMouseDown: execute { MAIN.Visualization.P14_CDISP.Active:=TRUE; }
        OnMouseUp: execute { MAIN.Visualization.P14_CDISP.Active:=FALSE; }
    Image (459,392 133x66), "%s", text variable: MAIN.Visualization.P14_CButton_9.display_text, invisible if: MAIN.Visualization.P14_CButton_9.invisible, image: ImagePool.PB_BU_160_75
        p84334746: MAIN.Visualization.P14_CButton_9.bitmap_ID
        OnMouseDown: execute { MAIN.Visualization.P14_CButton_9.Active:=TRUE; }
        OnMouseDown: write MAIN.Visualization.P14_Entered_trim via VisuDialogs.Numpad, min 10.0, max 44.0
        OnMouseUp: execute { MAIN.Visualization.P14_CButton_9.Active:=FALSE; }
    Image (597,392 133x66), "%s", text variable: MAIN.Visualization.P14_CButton_10.display_text, invisible if: MAIN.Visualization.P14_CButton_10.invisible, image: ImagePool.PB_BU_160_75
        p84334746: MAIN.Visualization.P14_CButton_10.bitmap_ID
        OnMouseDown: execute { MAIN.Visualization.P14_CButton_10.Active:=TRUE; }
        OnMouseDown: write MAIN.Visualization.P14_Entered_feed via VisuDialogs.Numpad, min 1.02, max 34.13
        OnMouseUp: execute { MAIN.Visualization.P14_CButton_10.Active:=FALSE; }
    Polyline (664,167) (684,157) (704,167) (694,187) (674,187), invisible if: MAIN.Visualization.P14_Profile.invisible
        p1285906596: MAIN.Visualization.P14_Profile_ARRAY_POINTER
    Polyline (661,262) (681,252) (701,262) (691,282) (671,282), invisible if: MAIN.Visualization.P14_HEAD.invisible
        p1285906596: MAIN.Visualization.P14_HEAD_ARRAY_POINTER
    Image (294,156 160x220), image: ImagePool.WELD_TOOL
        p84334746: MAIN.Visualization.P14_IMAGE.bitmap_ID
    Image (375,668 80x80), image: ImagePool.LJS
    Image (924,668 80x80), image: ImagePool.RJS
    Image (23,369 115x66), "%s", text variable: MAIN.Visualization.P14_CButton_2.display_text, invisible if: MAIN.Visualization.P14_CButton_2.invisible, image: ImagePool.PB_BU_75_75
        p84334746: MAIN.Visualization.P14_CButton_2.bitmap_ID
        OnMouseDown: execute { MAIN.Visualization.P14_CButton_2.Active:=TRUE; }
        OnMouseUp: execute { MAIN.Visualization.P14_CButton_2.Active:=FALSE; }
    Image (143,369 115x66), "%s", text variable: MAIN.Visualization.P14_CButton_4.display_text, invisible if: MAIN.Visualization.P14_CButton_4.invisible, image: ImagePool.PB_BU_75_75
        p84334746: MAIN.Visualization.P14_CButton_4.bitmap_ID
        OnMouseDown: execute { MAIN.Visualization.P14_CButton_4.Active:=TRUE; }
        OnMouseUp: execute { MAIN.Visualization.P14_CButton_4.Active:=FALSE; }
END_VISUALIZATION

(* stored: Version 1.1.0.1, ProductVersion 3.1.4022.12
   Visu TOOL_OPS_SCREEN: Id {95e9fb8a-502e-41f6-be3e-d4a9232d2c59} *)
